{attribute 'GeneratedUsingTerminal: EL2212-0000-0018'}
{attribute addProperty BoxType "EL2212-0000-0018"}
{attribute addProperty Id "DOX_Status_Channel_1AT %I*DOX_Status_Channel_09DD45C87DOX_Status_Channel_2AT %I*DOX_Status_Channel_09DD45C87DOX_Control_Channel_1AT %Q*DOX_Control_Channel_A74F23633DOX_Control_Channel_2AT %Q*DOX_Control_Channel_A74F23633WcStateAT %I*WcState_9091E0EB2InfoDataAT %I*InfoData_32EB74EA10"}
{attribute addProperty CRC "633081354"}
{attribute addProperty Size "32"}
TYPE EL2212_25BC0E0A EXTENDS EtcSlaveTerminalBase_947E5A46 :
STRUCT
	{attribute addProperty Name "DOX_Status_Channel_1"}
	DOX_Status_Channel_1 : DOX_Status_Channel_09DD45C8;
	{attribute addProperty Name "DOX_Status_Channel_2"}
	DOX_Status_Channel_2 : DOX_Status_Channel_09DD45C8;
	{attribute addProperty Name "DOX_Control_Channel_1"}
	DOX_Control_Channel_1 : DOX_Control_Channel_A74F2363;
	{attribute addProperty Name "DOX_Control_Channel_2"}
	DOX_Control_Channel_2 : DOX_Control_Channel_A74F2363;
	{attribute addProperty Name "WcState"}
	WcState : WcState_9091E0EB;
	{attribute addProperty Name "InfoData"}
	InfoData : InfoData_32EB74EA;
END_STRUCT
END_TYPE

(* stored: Version 1.2.0.0, ProductVersion 3.1.4024.9
   DUT EL2212_25BC0E0A: Id {7a25f223-8959-432f-a6bc-228ceb4188d9} *)
